// Mitsubishi GX Works2 project: klxsb   PLC: Q00J

// task Task_01 (event TRUE, interval 0, priority 31): POU_01

PROGRAM POU_01
klxsb:=X1;
END_PROGRAM
